{attribute 'no_explicit_call' := 'do not call this POU directly'}
{attribute 'hide_all_locals'}
FUNCTION_BLOCK INTERNAL FINAL FB_ArgumentsBuffer IMPLEMENTS I_ArgsBuffer

VAR
	aVarInputBuffer			: ARRAY [0..cMaxArgsBuffer - 1] OF BYTE;
	nVarInputBufferIndex	: UDINT := 0;
	aVarInputArgs			: ARRAY [0..cMaxArgs - 1] OF ST_AnyType;
	nVarInputIndex			: UDINT := 0;
	
	aVarInOutBuffer			: ARRAY [0..cMaxArgsBuffer - 1] OF BYTE;
	nVarInOutBufferIndex	: UDINT := 0;
	aAnyVarInOut			: ARRAY [0..cMaxArgs - 1] OF ST_AnyType;
	nAnyVarInOutIndex		: UDINT := 0;
	
	nRetValSizeTotal		: UDINT := 0;						// total size in Bytes of all In/Out arguments + return value
	stAnyRetVal				: ST_AnyType;
	
END_VAR

VAR CONSTANT
	cMaxArgsBuffer		: UDINT := Param_Args.cMaxArgsBuffer;	// max sizeof aArgs buffer array.
	cMaxArgs			: USINT := Param_Args.cMaxArgs;			// max length method arguments
END_VAR

METHOD GetRetVal : E_AdsErr
VAR_INPUT
END_VAR
VAR 
	i : UDINT;
	nLen : UDINT;
	pPtr : POINTER TO PVOID;
END_VAR
nVarInOutBufferIndex := 0;

IF stAnyRetVal.pValue <> NULL THEN
	nLen := TO_UDINT(stAnyRetVal.nSize);
	IF nLen > SIZEOF(aVarInOutBuffer) THEN
		GetRetVal := E_AdsErr.DEVICE_NOMEMORY;
		RETURN;
	END_IF
	MEMCPY(destAddr:= stAnyRetVal.pValue, srcAddr:= ADR(aVarInOutBuffer), n:= nLen);
	nVarInOutBufferIndex := nVarInOutBufferIndex + nLen;
END_IF


FOR i:=0 TO nAnyVarInOutIndex DO
	nLen := TO_UDINT(aAnyVarInOut[i].nSize);
	IF nLen + nVarInOutBufferIndex > SIZEOF(aVarInOutBuffer) THEN
		GetRetVal := E_AdsErr.DEVICE_NOMEMORY;
		RETURN;
	END_IF	
	IF aAnyVarInOut[i].TypeClass = __SYSTEM.TYPE_CLASS.TYPE_POINTER THEN
		pPtr := aAnyVarInOut[i].pValue;
		MEMCPY(destAddr:= pPtr^, srcAddr:= ADR(aVarInOutBuffer[nVarInOutBufferIndex]), n:= nLen);
	ELSE
		MEMCPY(destAddr:= aAnyVarInOut[i].pValue, srcAddr:= ADR(aVarInOutBuffer[nVarInOutBufferIndex]), n:= nLen);
	END_IF
	nVarInOutBufferIndex := nVarInOutBufferIndex + nLen;
END_FOR
END_METHOD

PROPERTY nArgsLength : UDINT
GET
nArgsLength := THIS^.nVarInputBufferIndex;
END_GET
END_PROPERTY

PROPERTY nRetValLength : UDINT
GET
nRetValLength := THIS^.nRetValSizeTotal;
END_GET
END_PROPERTY

PROPERTY pArgsBuffer : POINTER TO BYTE
GET
pArgsBuffer := ADR(aVarInputBuffer);
END_GET
END_PROPERTY

PROPERTY pRetValBuffer : POINTER TO BYTE
GET
pRetValBuffer := ADR(aVarInOutBuffer);
END_GET
END_PROPERTY

METHOD Reset
MEMSET(ADR(aVarInputBuffer), 16#0, SIZEOF(aVarInputBuffer));
MEMSET(ADR(aVarInputArgs), 16#0, SIZEOF(aVarInputArgs));
MEMSET(ADR(aVarInOutBuffer), 16#0, SIZEOF(aVarInOutBuffer));
MEMSET(ADR(aAnyVarInOut), 16#0, SIZEOF(aAnyVarInOut));
MEMSET(ADR(stAnyRetVal), 16#0, SIZEOF(stAnyRetVal));
nVarInputIndex := 0;
nVarInputBufferIndex := 0;
nVarInputBufferIndex := 0;
nAnyVarInOutIndex := 0;
nRetValSizeTotal := 0;
END_METHOD

METHOD SetRetVal
VAR_INPUT
	stAny : ST_AnyType;
END_VAR

stAnyRetVal := stAny;
nRetValSizeTotal := nRetValSizeTotal + TO_UDINT(stAny.nSize);
END_METHOD

METHOD SetVarInOut : E_AdsErr
VAR_INPUT
	stAny : ST_AnyType;
END_VAR
VAR
	eAdsErr : E_AdsErr;
END_VAR
IF stAny.pValue = NULL OR stAny.nSize <= 0 THEN
	SetVarInOut := E_AdsErr.DEVICE_INVALIDPARM;
	RETURN;
END_IF
IF nVarInOutBufferIndex + TO_UDINT(stAny.nSize) > SIZEOF(aVarInOutBuffer) THEN
	SetVarInOut := E_AdsErr.DEVICE_NOMEMORY;
	RETURN;
END_IF
IF nAnyVarInOutIndex > cMaxArgs -1  THEN
	SetVarInOut := E_AdsErr.DEVICE_NOMEMORY;
	RETURN;
END_IF

eAdsErr := SetVarInput(stAny);
IF eAdsErr <> E_AdsErr.NOERR THEN
	RETURN;
END_IF


aAnyVarInOut[nAnyVarInOutIndex] := stAny;
nAnyVarInOutIndex := nAnyVarInOutIndex + 1;
nRetValSizeTotal := nRetValSizeTotal + TO_UDINT(stAny.nSize);
END_METHOD

METHOD SetVarInput : E_AdsErr
VAR_INPUT
	stAny : ST_AnyType;
END_VAR
IF nVarInputBufferIndex + TO_UDINT(stAny.nSize) > SIZEOF(aVarInputBuffer) THEN
	SetVarInput := E_AdsErr.DEVICE_NOMEMORY;
	RETURN;
END_IF
IF nVarInputIndex > cMaxArgs -1  THEN
	SetVarInput := E_AdsErr.DEVICE_NOMEMORY;
	RETURN;
END_IF

aVarInputArgs[nVarInputIndex] := stAny;
nVarInputIndex := nVarInputIndex + 1;

MEMCPY(ADR(aVarInputBuffer[nVarInputBufferIndex]), stAny.pValue , TO_UDINT(stAny.nSize));
nVarInputBufferIndex := nVarInputBufferIndex + TO_UDINT(stAny.nSize);
END_METHOD

METHOD SetVarOutput : E_AdsErr
VAR_INPUT
	stAny : ST_AnyType;
END_VAR

IF stAny.pValue = NULL OR stAny.nSize <= 0 THEN
	SetVarOutput := E_AdsErr.DEVICE_INVALIDPARM;
	RETURN;
END_IF
IF nVarInOutBufferIndex + TO_UDINT(stAny.nSize) > SIZEOF(aVarInOutBuffer) THEN
	SetVarOutput := E_AdsErr.DEVICE_NOMEMORY;
	RETURN;
END_IF
IF nAnyVarInOutIndex > cMaxArgs -1  THEN
	SetVarOutput := E_AdsErr.DEVICE_NOMEMORY;
	RETURN;
END_IF


aAnyVarInOut[nAnyVarInOutIndex] := stAny;
nAnyVarInOutIndex := nAnyVarInOutIndex + 1;
nRetValSizeTotal := nRetValSizeTotal + TO_UDINT(stAny.nSize);
END_METHOD

END_FUNCTION_BLOCK

(* stored: Version 1.1.0.1, ProductVersion 3.1.4024.12
   POU FB_ArgumentsBuffer: Id {01fc2ce9-8258-4492-a9de-29c5e969f7ab}, SpecialFunc None
   Method GetRetVal: Id {cea3cce3-196b-409a-a8b2-458a46d7fe57}
   Property nArgsLength: Id {3e6406d3-8559-4369-8794-72dca5ed68cf}
   Get Get: Id {e52e01cc-4c3d-45ab-9d8c-cead13bb0390}
   Property nRetValLength: Id {10a70af2-342c-4cd7-a4b9-537f204ec7aa}
   Get Get: Id {bc8f807e-783a-40f3-87b0-5a44c6432025}
   Property pArgsBuffer: Id {c49081a2-557a-4182-8ca4-052eb5e6773a}
   Get Get: Id {67937687-456a-4488-99a4-7326b63d9c7e}
   Property pRetValBuffer: Id {56f5b221-f6a8-4b86-b562-294dbe5aec0f}
   Get Get: Id {784ee8ca-e535-4ada-90d4-785a8560acee}
   Method Reset: Id {4657a562-c23a-44ff-8c73-bd0243b995cf}
   Method SetRetVal: Id {39b01f18-bac1-4ecc-9b9c-1bb5c8a3f6d6}
   Method SetVarInOut: Id {d7cee7c5-ec2a-4636-8a08-f85c8fcac249}
   Method SetVarInput: Id {d617d063-fc4d-4b6f-8fcb-4090766deee1}
   Method SetVarOutput: Id {496fce22-2456-4b46-b473-18ca4e926a53} *)
